// TIA Portal project "S7-1500 için Lojik İşlem Komutları" (V18)

(* hardware
DEVICE "S7-1500/ET200MP station_1"  S7-1500 station
   slot 0: "Rail_0"  Rack  6ES7 590-1***0-0AA0
   slot 1: "PLC_1"  CPU 1512C-1 PN  6ES7 512-1CK00-0AB0  V2.8
      slot 3: "CPU display_1"  6ES7591-1AA00-0AA0
      slot 32768: "PROFINET interface_1"  X1
         slot 32769: "Port_1"  X1 P1
         slot 32770: "Port_2"  X1 P2
      slot 34817: "Virtual CP interface port_1"  Virtual CP interface port  Virtual CP interface port
*)

// ===== PLC "PLC_1"  CPU 1512C-1 PN =====

VAR_GLOBAL   // PLC tag table "Default tag table"
   "Tag_1" AT %I0.0 : Bool;
   "Tag_2" AT %MW10 : Int;
   "Tag_3" AT %Q0.0 : Bool;
   "Tag_4" AT %I0.1 : Bool;
   "Tag_5" AT %Q0.1 : Bool;
   "Tag_6" AT %MW11 : Int;
   "Tag_7" AT %MW12 : Int;
   "Tag_8" AT %MW13 : Int;
   "Tag_9" AT %MW14 : Int;
   "Tag_10" AT %I0.2 : Bool;
   "Tag_11" AT %I0.3 : Bool;
   "Tag_12" AT %MW5 : Word;
   "Tag_13" AT %MW6 : Word;
   "Tag_14" AT %MW8 : Word;
   "Tag_15" AT %MW19 : Word;
   "Tag_16" AT %MW9 : Word;
   "Tag_17" AT %M5.0 : Bool;
   "Tag_18" AT %Q0.2 : Bool;
   "Clock_Byte" AT %MB20 : Byte;
   "Clock_10Hz" AT %M20.0 : Bool;
   "Clock_5Hz" AT %M20.1 : Bool;
   "Clock_2.5Hz" AT %M20.2 : Bool;
   "Clock_2Hz" AT %M20.3 : Bool;
   "Clock_1.25Hz" AT %M20.4 : Bool;
   "Clock_1Hz" AT %M20.5 : Bool;
   "Clock_0.625Hz" AT %M20.6 : Bool;
   "Clock_0.5Hz" AT %M20.7 : Bool;
   "Tag_19" AT %M100.0 : Bool;
   "Tag_20" AT %QB0 : Byte;
   "Tag_21" AT %I0.4 : Bool;
   "Tag_22" AT %MW15 : Word;
END_VAR

// folder: System blocks/Program resources

DATA_BLOCK "IEC_Counter_0_DB"   // DB1
{ S7_Optimized_Access := 'TRUE' }
AUTHOR : Simatic
FAMILY : IEC
NAME : CNTR
VERSION : 1.0
// stored: InstanceOfName IEC_COUNTER
"IEC_COUNTER"
BEGIN
END_DATA_BLOCK

// folder: (top level)

ORGANIZATION_BLOCK "Main"   // OB1, LAD, ProgramCycle
TITLE = "Main Program Sweep (Cycle)"
{ S7_Optimized_Access := 'TRUE' }
VERSION : 0.1
   VAR_INPUT
      Initial_Call : Bool;   // Initial call of this OB
      Remanence : Bool;   // =True, if remanent data are available
   END_VAR
BEGIN

REGION Network 1: Toplama İlemi(ADD)
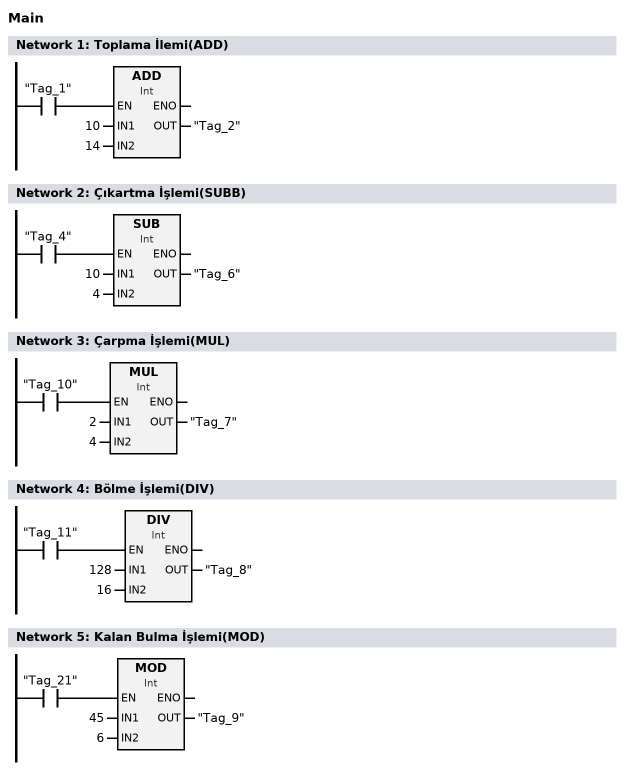
   RUNG wire#powerrail
      Contact( "Tag_1" )
      { S7_Templates := "SrcType := Int" } Add(in1 := 10, in2 := 14, out => "Tag_2")
   END_RUNG
   // the same network as SCL:
   IF "Tag_1" THEN "Tag_2" := 10 + 14; END_IF;
END_REGION

REGION Network 2: Çıkartma İşlemi(SUBB)
   RUNG wire#powerrail
      Contact( "Tag_4" )
      { S7_Templates := "SrcType := Int" } Sub(in1 := 10, in2 := 4, out => "Tag_6")
   END_RUNG
   // the same network as SCL:
   IF "Tag_4" THEN "Tag_6" := 10 - 4; END_IF;
END_REGION

REGION Network 3: Çarpma İşlemi(MUL)
   RUNG wire#powerrail
      Contact( "Tag_10" )
      { S7_Templates := "SrcType := Int" } Mul(in1 := 2, in2 := 4, out => "Tag_7")
   END_RUNG
   // the same network as SCL:
   IF "Tag_10" THEN "Tag_7" := 2 * 4; END_IF;
END_REGION

REGION Network 4: Bölme İşlemi(DIV)
   RUNG wire#powerrail
      Contact( "Tag_11" )
      { S7_Templates := "SrcType := Int" } Div(in1 := 128, in2 := 16, out => "Tag_8")
   END_RUNG
   // the same network as SCL:
   IF "Tag_11" THEN "Tag_8" := 128 / 16; END_IF;
END_REGION

REGION Network 5: Kalan Bulma İşlemi(MOD)
   RUNG wire#powerrail
      Contact( "Tag_21" )
      { S7_Templates := "SrcType := Int" } Mod(in1 := 45, in2 := 6, out => "Tag_9")
   END_RUNG
   // the same network as SCL:
   IF "Tag_21" THEN "Tag_9" := 45 MOD 6; END_IF;
END_REGION
END_ORGANIZATION_BLOCK